PROGRAM Motion
VAR
	FB_Power: MC_Power;
	FB_Stop: MC_Stop;
	FB_Velocity: MC_MoveVelocity;
	FB_Relative: MC_MoveRelative;
	FB_ReadStatus: MC_ReadStatus;

	
END_VAR

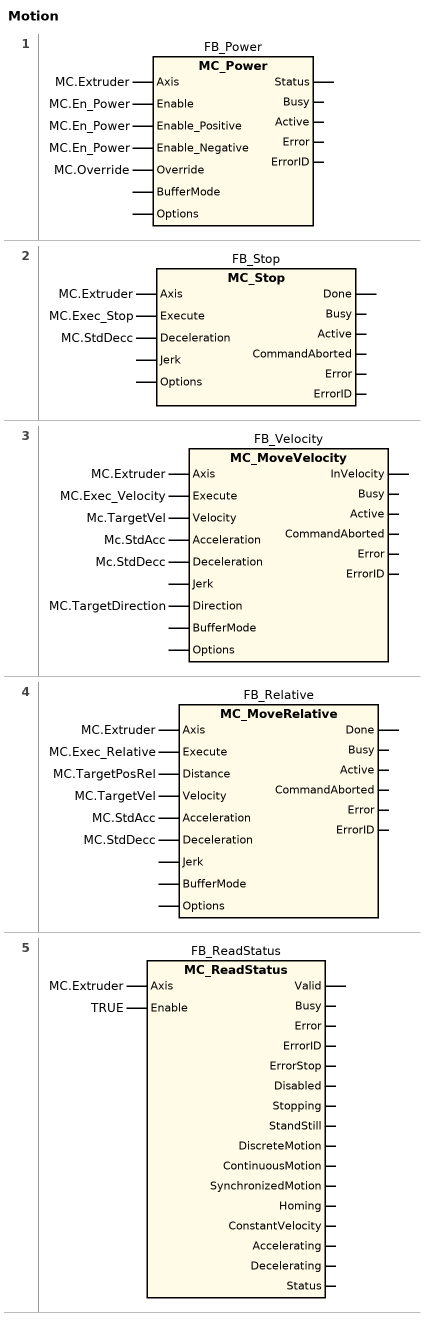
// NETWORK 1
FB_Power(
    Axis := MC.Extruder,
    Enable := MC.En_Power,
    Enable_Positive := MC.En_Power,
    Enable_Negative := MC.En_Power,
    Override := MC.Override); // MC_Power

// NETWORK 2
FB_Stop(Axis := MC.Extruder, Execute := MC.Exec_Stop, Deceleration := MC.StdDecc); // MC_Stop

// NETWORK 3
FB_Velocity(
    Axis := MC.Extruder,
    Execute := MC.Exec_Velocity,
    Velocity := Mc.TargetVel,
    Acceleration := Mc.StdAcc,
    Deceleration := Mc.StdDecc,
    Direction := MC.TargetDirection); // MC_MoveVelocity

// NETWORK 4
FB_Relative(
    Axis := MC.Extruder,
    Execute := MC.Exec_Relative,
    Distance := MC.TargetPosRel,
    Velocity := MC.TargetVel,
    Acceleration := MC.StdAcc,
    Deceleration := MC.StdDecc); // MC_MoveRelative

// NETWORK 5
FB_ReadStatus(Axis := MC.Extruder, Enable := TRUE); // MC_ReadStatus

ACTION InitMotion:
Mc.En_Power := FALSE;
MC.Exec_Relative := FALSE;
MC.Exec_Stop := FALSE;
MC.Exec_Velocity := FALSE;
END_ACTION

END_PROGRAM

(* stored: Version 1.1.0.1, ProductVersion 3.1.4024.9
   POU Motion: Id {d206c616-e0b3-44bf-898b-092307161bef}, SpecialFunc None
   Action InitMotion: Id {9d46ed5d-55f9-4643-b0b6-d4b7f5e5ed0d} *)
